TYPE EtcSlaveBase_82538BE2 :
STRUCT
END_STRUCT
END_TYPE

(* stored: Version 1.2.0.0, ProductVersion 3.1.4024.11
   DUT EtcSlaveBase_82538BE2: Id {3e940d06-9758-4fbf-9b38-b7c79233bf1d} *)
